(* CoDeSys 2.3 export: FB_WHEELCHAIRLIFTLIMIT.EXP *)

(* POU 4_DoorFunctions/FB_wheelchairliftlimit, LD *)
FUNCTION_BLOCK FB_wheelchairliftlimit
VAR_INPUT
	dooropen						:BOOL;
	doorspread					:BOOL;
END_VAR
VAR_OUTPUT
	wheelchairliftlimitOK			:BOOL
END_VAR
VAR
END_VAR
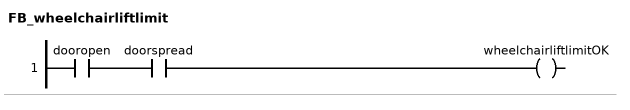
_LD_ (* Ladder Diagram *)
NETWORK 1
	[dooropen] - [doorspread] --- (wheelchairliftlimitOK)
_END_LD_
(* the same logic as Structured Text *)
(* Network 1 *)
wheelchairliftlimitOK := dooropen AND doorspread;
END_FUNCTION_BLOCK
